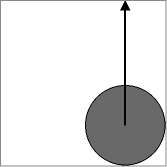
VISUALIZATION VISU_Tube_Top_0  // 167x167
VAR_IN_OUT
	azi : LREAL;
END_VAR
    Ellipse (85,85 80x80)
        p2858320360: azi
    Polygon (120,10) (125,0) (130,10)
        p2858320360: azi
    Polyline (125,125) (125,10)
        p2858320360: azi
END_VISUALIZATION

(* stored: Version 1.1.0.1, ProductVersion 3.1.4018.5
   Visu VISU_Tube_Top_0: Id {3fcab3be-727c-439a-9665-07054bb827bf} *)
